// TIA Portal V16 export
// export: Created 2025-10-06T17:54:37.2631868Z, ExportSetting WithDefaults, DisplayName Totally Integrated Automation Portal, DisplayVersion V16, DisplayName TIA Portal Version Control Interface, DisplayVersion V16, DisplayName TIA Portal Openness, DisplayVersion V16, DisplayName STEP 7 Professional, DisplayVersion V16, DisplayName STEP 7 Safety, DisplayVersion V16, DisplayName WinCC Advanced, DisplayVersion V16
DATA_BLOCK "IEC_Timer_0_DB"   // DB31
// stored: AutoNumber true, InstanceOfName TON_SFB, OfSystemLibElement TON, OfSystemLibVersion 1.0
"TON_SFB"
   // VAR_INPUT
   //    IN : Bool;
   //    PT : Time;
   // END_VAR
   // VAR_OUTPUT
   //    Q : Bool;
   //    ET : Time;
   // END_VAR
   // VAR RETAIN
   //    STATE : Byte;
   //    STIME : Time;
   //    ATIME : Time;
   // END_VAR
BEGIN
END_DATA_BLOCK
